// TwinCAT 3 PLC project lamp_lv17_motion
// ProgramVersion: 3.1.4022.7
// libraries:
//   Tc2_MC2, * (Beckhoff Automation GmbH)
//   Tc2_Standard, * (Beckhoff Automation GmbH)
//   Tc2_System, * (Beckhoff Automation GmbH)
//   Tc2_Utilities, * (Beckhoff Automation GmbH)
//   Tc3_Module, * (Beckhoff Automation GmbH)
//   lcls-twincat-motion,newest,SLAC
// project tree:
//   / PlcTask.TcTTO (not stored)
//   POUs/ Main.TcPOU
// real-time tasks:
//   TASK PlcTask: cycle T#10ms, priority 20, ADS port 350
// motion (NC):
//   TASK NC-Task 1 SAF: cycle T#2ms, priority 4, ADS port 501
//   TASK NC-Task 1 SVB: cycle T#10ms, priority 8, ADS port 511
//   AXIS GasJetX (id 1)
//   AXIS GasJetY (id 2)
//   AXIS GasJetZ (id 3)
//   AXIS SamplePaddleX (id 4)
//     Dynamic: Acceleration=2, Deceleration=2, DelayTime=0.008
//     Velo: Maximum=1
//     TargetPosControl: Range=0.001, Time=0.1
//     OtherSettings: AllowMotionCmdToSlave=true
//     encoder EncType=4
//       EncPara: ScaleFactorNumerator=1e-05, Inverse=true, MaxCount=#xffffffff
//         SoftEndMinControl: Range=-39
//         Inc: RefSoftSyncMask=#x0000ffff
//     drive DrvType=24
//       DrvPara: Inverse=true
//         Analog: VeloReferenz=10, ScaleFactorActTorque=0.1
//         TimeComp: TaskDelayCycles=1
//     controller CtrType=2
//       CtrPara: PriorControlFactor=1
//         PosDiffControl: Range=1
//         PID: PosKp=20, PosExtKp=50, DeadBandPosition=0.0005
//         Observer: BandWidth=20
//   AXIS SamplePaddleY (id 5)
//     Dynamic: Acceleration=2, Deceleration=2, DelayTime=0.008
//     Velo: Maximum=1
//     TargetPosControl: Range=0.01, Time=0.1
//     OtherSettings: AllowMotionCmdToSlave=true
//     encoder EncType=4
//       EncPara: ScaleFactorNumerator=2e-05, Inverse=true, MaxCount=#xffffffff
//         SoftEndMinControl: Range=-10
//         SoftEndMaxControl: Range=10
//         Inc: RefSoftSyncMask=#x0000ffff
//     drive DrvType=24
//       DrvPara: Inverse=true
//         Analog: VeloReferenz=5, ScaleFactorActTorque=0.1
//         TimeComp: TaskDelayCycles=1
//     controller CtrType=2
//       CtrPara: PriorControlFactor=1
//         PosDiffControl: Range=0.5
//         PID: PosKp=40, PosExtKp=75, DeadBandPosition=0.0005
//         Observer: BandWidth=20
//   AXIS SamplePaddleZ (id 6)
//     Dynamic: Acceleration=2, Deceleration=2, DelayTime=0.008
//     Velo: Maximum=1
//     TargetPosControl: Range=0.001, Time=0.1
//     OtherSettings: AllowMotionCmdToSlave=true
//     encoder EncType=4
//       EncPara: ScaleFactorNumerator=1e-05, Inverse=true, MaxCount=#xffffffff
//         Inc: RefSoftSyncMask=#x0000ffff
//     drive DrvType=24
//       DrvPara: Inverse=true
//         Analog: VeloReferenz=10, ScaleFactorActTorque=0.1
//         TimeComp: TaskDelayCycles=1
//     controller CtrType=2
//       CtrPara: PriorControlFactor=1
//         PosDiffControl: Range=1
//         PID: PosKp=20, PosExtKp=50, DeadBandPosition=0.0005
//         Observer: BandWidth=20
//   AXIS DetectorX (id 7)
//     Dynamic: Acceleration=2, Deceleration=2
//     Velo: Maximum=1
//     TargetPosControl: Range=0.001
//     OtherSettings: AllowMotionCmdToSlave=true
//     encoder EncType=4
//       EncPara: ScaleFactorNumerator=7.8125e-05, Inverse=true, MaxCount=#x0000ffff
//         Inc: RefSoftSyncMask=#x0000ffff
//     drive DrvType=24
//       DrvPara: Inverse=true
//         Analog: VeloReferenz=10, ScaleFactorActTorque=0.1
//         TimeComp: TaskDelayCycles=1
//     controller CtrType=2
//       CtrPara: PriorControlFactor=1
//         PosDiffControl: Range=1
//         PID: PosKp=20, PosExtKp=50, DeadBandPosition=0.0005
//         Observer: BandWidth=20
//   AXIS DetectorY (id 8)
//     Dynamic: Acceleration=2, Deceleration=2
//     Velo: Maximum=1
//     TargetPosControl: Range=0.001
//     OtherSettings: AllowMotionCmdToSlave=true
//     encoder EncType=4
//       EncPara: ScaleFactorNumerator=7.8125e-05, MaxCount=#x0000ffff
//         Inc: RefSoftSyncMask=#x0000ffff
//     drive DrvType=24
//       Analog: VeloReferenz=10, ScaleFactorActTorque=0.1
//       TimeComp: TaskDelayCycles=1
//     controller CtrType=2
//       CtrPara: PriorControlFactor=1
//         PosDiffControl: Range=1
//         PID: PosKp=20, PosExtKp=50, DeadBandPosition=0.0005
//         Observer: BandWidth=20
// I/O:
//   DEVICE PLC Rail (EtherCAT)
// variable links:
//   (this object) <-> PLC Rail (EtherCAT)/Power (EK1200)/PLC Junction 1 (EK1122)/X1 VacuumMotion (EK1100)/SamplePaddleX-Enc-EL5021
//     Enc/Inputs/In/nDataIn1 <-> ENC Status/Counter value
//     Enc/Inputs/In/nDataIn2 <-> ENC Status/Latch value
//     Enc/Inputs/In/nState1 <-> ENC Status/Status/Latch C valid
//     Enc/Inputs/In/nState1 @bit 2 <-> ENC Status/Status/Set counter done
//     Enc/Inputs/In/nState2 @bit 2 <-> ENC Status/Status/Status of input C
//     Enc/Inputs/In/nState2 @bit 5 <-> ENC Status/Status/Sync error
//     Enc/Inputs/In/nState2 @bit 6 <-> ENC Status/Status/TxPDO State
//     Enc/Inputs/In/nState2 @bit 7 <-> ENC Status/Status/TxPDO Toggle
//     Enc/Inputs/In/nState3 @bit 4 <-> ENC Status/Status/Amplitude error
//     Enc/Inputs/In/nState3 @bit 3 <-> ENC Status/Status/Frequency error
//     Enc/Inputs/In/nState4 @bit 1 <-> WcState/InputToggle
//     Enc/Inputs/In/nState4 <-> WcState/WcState
//     Enc/Outputs/Out/nCtrl1 <-> ENC Control/Control/Enable latch C
//     Enc/Outputs/Out/nCtrl1 @bit 2 <-> ENC Control/Control/Set counter
//     Enc/Outputs/Out/nDataOut1 <-> ENC Control/Set counter value
//   (this object) <-> PLC Rail (EtherCAT)/Power (EK1200)/PLC Junction 1 (EK1122)/X1 VacuumMotion (EK1100)/SamplePaddleX-Mot-EL7041
//     Drive/Inputs/In/nState1 @bit 3 <-> STM Status/Status/Error
//     Drive/Inputs/In/nState1 @bit 5 <-> STM Status/Status/Moving negative
//     Drive/Inputs/In/nState1 @bit 4 <-> STM Status/Status/Moving positive
//     Drive/Inputs/In/nState1 @bit 1 <-> STM Status/Status/Ready
//     Drive/Inputs/In/nState1 <-> STM Status/Status/Ready to enable
//     Drive/Inputs/In/nState1 @bit 6 <-> STM Status/Status/Torque reduced
//     Drive/Inputs/In/nState1 @bit 2 <-> STM Status/Status/Warning
//     Drive/Inputs/In/nState2 @bit 3 <-> STM Status/Status/Digital input 1
//     Drive/Inputs/In/nState2 @bit 4 <-> STM Status/Status/Digital input 2
//     Drive/Inputs/In/nState2 @bit 5 <-> STM Status/Status/Sync error
//     Drive/Inputs/In/nState2 @bit 7 <-> STM Status/Status/TxPDO Toggle
//     Drive/Inputs/In/nState4 @bit 1 <-> WcState/InputToggle
//     Drive/Inputs/In/nState4 <-> WcState/WcState
//     Drive/Outputs/Out/nCtrl1 <-> STM Control/Control/Enable
//     Drive/Outputs/Out/nCtrl1 @bit 2 <-> STM Control/Control/Reduce torque
//     Drive/Outputs/Out/nCtrl1 @bit 1 <-> STM Control/Control/Reset
//     Drive/Outputs/Out/nDataOut2[0] <-> STM Velocity/Velocity
//   (this object) <-> PLC Rail (EtherCAT)/Power (EK1200)/PLC Junction 1 (EK1122)/X1 VacuumMotion (EK1100)/SamplePaddleY-Enc-EL5021
//     Enc/Inputs/In/nDataIn1 <-> ENC Status/Counter value
//     Enc/Inputs/In/nDataIn2 <-> ENC Status/Latch value
//     Enc/Inputs/In/nState1 <-> ENC Status/Status/Latch C valid
//     Enc/Inputs/In/nState1 @bit 2 <-> ENC Status/Status/Set counter done
//     Enc/Inputs/In/nState2 @bit 2 <-> ENC Status/Status/Status of input C
//     Enc/Inputs/In/nState2 @bit 5 <-> ENC Status/Status/Sync error
//     Enc/Inputs/In/nState2 @bit 6 <-> ENC Status/Status/TxPDO State
//     Enc/Inputs/In/nState2 @bit 7 <-> ENC Status/Status/TxPDO Toggle
//     Enc/Inputs/In/nState3 @bit 4 <-> ENC Status/Status/Amplitude error
//     Enc/Inputs/In/nState3 @bit 3 <-> ENC Status/Status/Frequency error
//     Enc/Inputs/In/nState4 @bit 1 <-> WcState/InputToggle
//     Enc/Inputs/In/nState4 <-> WcState/WcState
//     Enc/Outputs/Out/nCtrl1 <-> ENC Control/Control/Enable latch C
//     Enc/Outputs/Out/nCtrl1 @bit 2 <-> ENC Control/Control/Set counter
//     Enc/Outputs/Out/nDataOut1 <-> ENC Control/Set counter value
//   (this object) <-> PLC Rail (EtherCAT)/Power (EK1200)/PLC Junction 1 (EK1122)/X1 VacuumMotion (EK1100)/SamplePaddleY-Mot-EL7041
//     Drive/Inputs/In/nState1 @bit 3 <-> STM Status/Status/Error
//     Drive/Inputs/In/nState1 @bit 5 <-> STM Status/Status/Moving negative
//     Drive/Inputs/In/nState1 @bit 4 <-> STM Status/Status/Moving positive
//     Drive/Inputs/In/nState1 @bit 1 <-> STM Status/Status/Ready
//     Drive/Inputs/In/nState1 <-> STM Status/Status/Ready to enable
//     Drive/Inputs/In/nState1 @bit 6 <-> STM Status/Status/Torque reduced
//     Drive/Inputs/In/nState1 @bit 2 <-> STM Status/Status/Warning
//     Drive/Inputs/In/nState2 @bit 3 <-> STM Status/Status/Digital input 1
//     Drive/Inputs/In/nState2 @bit 4 <-> STM Status/Status/Digital input 2
//     Drive/Inputs/In/nState2 @bit 5 <-> STM Status/Status/Sync error
//     Drive/Inputs/In/nState2 @bit 7 <-> STM Status/Status/TxPDO Toggle
//     Drive/Inputs/In/nState4 @bit 1 <-> WcState/InputToggle
//     Drive/Inputs/In/nState4 <-> WcState/WcState
//     Drive/Outputs/Out/nCtrl1 <-> STM Control/Control/Enable
//     Drive/Outputs/Out/nCtrl1 @bit 2 <-> STM Control/Control/Reduce torque
//     Drive/Outputs/Out/nCtrl1 @bit 1 <-> STM Control/Control/Reset
//     Drive/Outputs/Out/nDataOut2[0] <-> STM Velocity/Velocity
//   (this object) <-> PLC Rail (EtherCAT)/Power (EK1200)/PLC Junction 1 (EK1122)/X1 VacuumMotion (EK1100)/SamplePaddleZ-Enc-EL5021
//     Enc/Inputs/In/nDataIn1 <-> ENC Status/Counter value
//     Enc/Inputs/In/nDataIn2 <-> ENC Status/Latch value
//     Enc/Inputs/In/nState1 <-> ENC Status/Status/Latch C valid
//     Enc/Inputs/In/nState1 @bit 2 <-> ENC Status/Status/Set counter done
//     Enc/Inputs/In/nState2 @bit 2 <-> ENC Status/Status/Status of input C
//     Enc/Inputs/In/nState2 @bit 5 <-> ENC Status/Status/Sync error
//     Enc/Inputs/In/nState2 @bit 6 <-> ENC Status/Status/TxPDO State
//     Enc/Inputs/In/nState2 @bit 7 <-> ENC Status/Status/TxPDO Toggle
//     Enc/Inputs/In/nState3 @bit 4 <-> ENC Status/Status/Amplitude error
//     Enc/Inputs/In/nState3 @bit 3 <-> ENC Status/Status/Frequency error
//     Enc/Inputs/In/nState4 @bit 1 <-> WcState/InputToggle
//     Enc/Inputs/In/nState4 <-> WcState/WcState
//     Enc/Outputs/Out/nCtrl1 <-> ENC Control/Control/Enable latch C
//     Enc/Outputs/Out/nCtrl1 @bit 2 <-> ENC Control/Control/Set counter
//     Enc/Outputs/Out/nDataOut1 <-> ENC Control/Set counter value
//   (this object) <-> PLC Rail (EtherCAT)/Power (EK1200)/PLC Junction 1 (EK1122)/X1 VacuumMotion (EK1100)/SamplePaddleZ-Mot-EL7041
//     Drive/Inputs/In/nState1 @bit 3 <-> STM Status/Status/Error
//     Drive/Inputs/In/nState1 @bit 5 <-> STM Status/Status/Moving negative
//     Drive/Inputs/In/nState1 @bit 4 <-> STM Status/Status/Moving positive
//     Drive/Inputs/In/nState1 @bit 1 <-> STM Status/Status/Ready
//     Drive/Inputs/In/nState1 <-> STM Status/Status/Ready to enable
//     Drive/Inputs/In/nState1 @bit 6 <-> STM Status/Status/Torque reduced
//     Drive/Inputs/In/nState1 @bit 2 <-> STM Status/Status/Warning
//     Drive/Inputs/In/nState2 @bit 3 <-> STM Status/Status/Digital input 1
//     Drive/Inputs/In/nState2 @bit 4 <-> STM Status/Status/Digital input 2
//     Drive/Inputs/In/nState2 @bit 5 <-> STM Status/Status/Sync error
//     Drive/Inputs/In/nState2 @bit 7 <-> STM Status/Status/TxPDO Toggle
//     Drive/Inputs/In/nState4 @bit 1 <-> WcState/InputToggle
//     Drive/Inputs/In/nState4 <-> WcState/WcState
//     Drive/Outputs/Out/nCtrl1 <-> STM Control/Control/Enable
//     Drive/Outputs/Out/nCtrl1 @bit 2 <-> STM Control/Control/Reduce torque
//     Drive/Outputs/Out/nCtrl1 @bit 1 <-> STM Control/Control/Reset
//     Drive/Outputs/Out/nDataOut2[0] <-> STM Velocity/Velocity
//   (this object) <-> PLC Rail (EtherCAT)/Power (EK1200)/PLC Junction 1 (EK1122)/X1 VacuumMotion (EK1100)/DetectorX-Mot-EL7041
//     Drive/Inputs/In/nState1 @bit 3 <-> STM Status/Status/Error
//     Drive/Inputs/In/nState1 @bit 5 <-> STM Status/Status/Moving negative
//     Drive/Inputs/In/nState1 @bit 4 <-> STM Status/Status/Moving positive
//     Drive/Inputs/In/nState1 @bit 1 <-> STM Status/Status/Ready
//     Drive/Inputs/In/nState1 <-> STM Status/Status/Ready to enable
//     Drive/Inputs/In/nState1 @bit 6 <-> STM Status/Status/Torque reduced
//     Drive/Inputs/In/nState1 @bit 2 <-> STM Status/Status/Warning
//     Drive/Inputs/In/nState2 @bit 3 <-> STM Status/Status/Digital input 1
//     Drive/Inputs/In/nState2 @bit 4 <-> STM Status/Status/Digital input 2
//     Drive/Inputs/In/nState2 @bit 5 <-> STM Status/Status/Sync error
//     Drive/Inputs/In/nState2 @bit 7 <-> STM Status/Status/TxPDO Toggle
//     Drive/Inputs/In/nState4 @bit 1 <-> WcState/InputToggle
//     Drive/Inputs/In/nState4 <-> WcState/WcState
//     Drive/Outputs/Out/nCtrl1 <-> STM Control/Control/Enable
//     Drive/Outputs/Out/nCtrl1 @bit 2 <-> STM Control/Control/Reduce torque
//     Drive/Outputs/Out/nCtrl1 @bit 1 <-> STM Control/Control/Reset
//     Drive/Outputs/Out/nDataOut2[0] <-> STM Velocity/Velocity
//     Enc/Inputs/In/nDataIn1[0] <-> ENC Status compact/Counter value
//     Enc/Inputs/In/nDataIn2[0] <-> ENC Status compact/Latch value
//     Enc/Inputs/In/nState1 @bit 4 <-> ENC Status compact/Status/Counter overflow
//     Enc/Inputs/In/nState1 @bit 3 <-> ENC Status compact/Status/Counter underflow
//     Enc/Inputs/In/nState1 @bit 7 <-> ENC Status compact/Status/Extrapolation stall
//     Enc/Inputs/In/nState1 <-> ENC Status compact/Status/Latch C valid
//     Enc/Inputs/In/nState1 @bit 1 <-> ENC Status compact/Status/Latch extern valid
//     Enc/Inputs/In/nState1 @bit 2 <-> ENC Status compact/Status/Set counter done
//     Enc/Inputs/In/nState2 @bit 4 <-> ENC Status compact/Status/Status of extern latch
//     Enc/Inputs/In/nState2 <-> ENC Status compact/Status/Status of input A
//     Enc/Inputs/In/nState2 @bit 1 <-> ENC Status compact/Status/Status of input B
//     Enc/Inputs/In/nState2 @bit 2 <-> ENC Status compact/Status/Status of input C
//     Enc/Inputs/In/nState2 @bit 5 <-> ENC Status compact/Status/Sync error
//     Enc/Inputs/In/nState2 @bit 7 <-> ENC Status compact/Status/TxPDO Toggle
//     Enc/Inputs/In/nState4 @bit 1 <-> WcState/InputToggle
//     Enc/Inputs/In/nState4 <-> WcState/WcState
//     Enc/Outputs/Out/nCtrl1 <-> ENC Control compact/Control/Enable latch C
//     Enc/Outputs/Out/nCtrl1 @bit 3 <-> ENC Control compact/Control/Enable latch extern on negative edge
//     Enc/Outputs/Out/nCtrl1 @bit 1 <-> ENC Control compact/Control/Enable latch extern on positive edge
//     Enc/Outputs/Out/nCtrl1 @bit 2 <-> ENC Control compact/Control/Set counter
//     Enc/Outputs/Out/nDataOut1[0] <-> ENC Control compact/Set counter value
//   (this object) <-> PLC Rail (EtherCAT)/Power (EK1200)/PLC Junction 1 (EK1122)/X1 VacuumMotion (EK1100)/DetectorY-Mot-EL7041
//     Drive/Inputs/In/nState1 @bit 3 <-> STM Status/Status/Error
//     Drive/Inputs/In/nState1 @bit 5 <-> STM Status/Status/Moving negative
//     Drive/Inputs/In/nState1 @bit 4 <-> STM Status/Status/Moving positive
//     Drive/Inputs/In/nState1 @bit 1 <-> STM Status/Status/Ready
//     Drive/Inputs/In/nState1 <-> STM Status/Status/Ready to enable
//     Drive/Inputs/In/nState1 @bit 6 <-> STM Status/Status/Torque reduced
//     Drive/Inputs/In/nState1 @bit 2 <-> STM Status/Status/Warning
//     Drive/Inputs/In/nState2 @bit 3 <-> STM Status/Status/Digital input 1
//     Drive/Inputs/In/nState2 @bit 4 <-> STM Status/Status/Digital input 2
//     Drive/Inputs/In/nState2 @bit 5 <-> STM Status/Status/Sync error
//     Drive/Inputs/In/nState2 @bit 7 <-> STM Status/Status/TxPDO Toggle
//     Drive/Inputs/In/nState4 @bit 1 <-> WcState/InputToggle
//     Drive/Inputs/In/nState4 <-> WcState/WcState
//     Drive/Outputs/Out/nCtrl1 <-> STM Control/Control/Enable
//     Drive/Outputs/Out/nCtrl1 @bit 2 <-> STM Control/Control/Reduce torque
//     Drive/Outputs/Out/nCtrl1 @bit 1 <-> STM Control/Control/Reset
//     Drive/Outputs/Out/nDataOut2[0] <-> STM Velocity/Velocity
//     Enc/Inputs/In/nDataIn1[0] <-> ENC Status compact/Counter value
//     Enc/Inputs/In/nDataIn2[0] <-> ENC Status compact/Latch value
//     Enc/Inputs/In/nState1 @bit 4 <-> ENC Status compact/Status/Counter overflow
//     Enc/Inputs/In/nState1 @bit 3 <-> ENC Status compact/Status/Counter underflow
//     Enc/Inputs/In/nState1 @bit 7 <-> ENC Status compact/Status/Extrapolation stall
//     Enc/Inputs/In/nState1 <-> ENC Status compact/Status/Latch C valid
//     Enc/Inputs/In/nState1 @bit 1 <-> ENC Status compact/Status/Latch extern valid
//     Enc/Inputs/In/nState1 @bit 2 <-> ENC Status compact/Status/Set counter done
//     Enc/Inputs/In/nState2 @bit 4 <-> ENC Status compact/Status/Status of extern latch
//     Enc/Inputs/In/nState2 <-> ENC Status compact/Status/Status of input A
//     Enc/Inputs/In/nState2 @bit 1 <-> ENC Status compact/Status/Status of input B
//     Enc/Inputs/In/nState2 @bit 2 <-> ENC Status compact/Status/Status of input C
//     Enc/Inputs/In/nState2 @bit 5 <-> ENC Status compact/Status/Sync error
//     Enc/Inputs/In/nState2 @bit 7 <-> ENC Status compact/Status/TxPDO Toggle
//     Enc/Inputs/In/nState4 @bit 1 <-> WcState/InputToggle
//     Enc/Inputs/In/nState4 <-> WcState/WcState
//     Enc/Outputs/Out/nCtrl1 <-> ENC Control compact/Control/Enable latch C
//     Enc/Outputs/Out/nCtrl1 @bit 3 <-> ENC Control compact/Control/Enable latch extern on negative edge
//     Enc/Outputs/Out/nCtrl1 @bit 1 <-> ENC Control compact/Control/Enable latch extern on positive edge
//     Enc/Outputs/Out/nCtrl1 @bit 2 <-> ENC Control compact/Control/Set counter
//     Enc/Outputs/Out/nDataOut1[0] <-> ENC Control compact/Set counter value
//   lamp_lv17_motion Instance <-> PLC Rail (EtherCAT)/Power (EK1200)/PLC Junction 1 (EK1122)/X1 AtmosphereMotion (EK1100)/GasJetX-EL7041
//     PlcTask Inputs/Main.M1.bLimitBackwardEnable <-> STM Status/Status/Digital input 2
//     PlcTask Inputs/Main.M1.bLimitForwardEnable <-> STM Status/Status/Digital input 1
//   lamp_lv17_motion Instance <-> PLC Rail (EtherCAT)/Power (EK1200)/PLC Junction 1 (EK1122)/X1 AtmosphereMotion (EK1100)/GasJetY-EL7041
//     PlcTask Inputs/Main.M2.bLimitBackwardEnable <-> STM Status/Status/Digital input 2
//     PlcTask Inputs/Main.M2.bLimitForwardEnable <-> STM Status/Status/Digital input 1
//   lamp_lv17_motion Instance <-> PLC Rail (EtherCAT)/Power (EK1200)/PLC Junction 1 (EK1122)/X1 AtmosphereMotion (EK1100)/GasJetZ-EL7041
//     PlcTask Inputs/Main.M3.bLimitBackwardEnable <-> STM Status/Status/Digital input 2
//     PlcTask Inputs/Main.M3.bLimitForwardEnable <-> STM Status/Status/Digital input 1
//   lamp_lv17_motion Instance <-> PLC Rail (EtherCAT)/Power (EK1200)/PLC Junction 1 (EK1122)/X1 VacuumMotion (EK1100)/DetectorXY-Limits-EL1084
//     PlcTask Inputs/Main.M7.bLimitBackwardEnable <-> Channel 2/Input
//     PlcTask Inputs/Main.M8.bLimitBackwardEnable <-> Channel 4/Input
//     PlcTask Inputs/Main.M7.bLimitForwardEnable <-> Channel 1/Input
//   lamp_lv17_motion Instance <-> PLC Rail (EtherCAT)/Power (EK1200)/PLC Junction 1 (EK1122)/X1 VacuumMotion (EK1100)/SamplePaddleXY-Limits-EL1084
//     PlcTask Inputs/Main.M4.bLimitBackwardEnable <-> Channel 2/Input
//     PlcTask Inputs/Main.M5.bLimitBackwardEnable <-> Channel 3/Input
//     PlcTask Inputs/Main.M4.bLimitForwardEnable <-> Channel 1/Input
//     PlcTask Inputs/Main.M5.bLimitForwardEnable <-> Channel 4/Input
//   lamp_lv17_motion Instance <-> PLC Rail (EtherCAT)/Power (EK1200)/PLC Junction 1 (EK1122)/X1 VacuumMotion (EK1100)/SamplePaddleZ-Limits-EL1084
//     PlcTask Inputs/Main.M6.bLimitBackwardEnable <-> Channel 2/Input
//     PlcTask Inputs/Main.M6.bLimitForwardEnable <-> Channel 1/Input
//   lamp_lv17_motion Instance <-> NC-Task 1 SAF/Axes/DetectorX
//     PlcTask Inputs/Main.M7.Axis.NcToPlc <-> Outputs/ToPlc
//     PlcTask Outputs/Main.M7.Axis.PlcToNc <-> Inputs/FromPlc
//   lamp_lv17_motion Instance <-> NC-Task 1 SAF/Axes/DetectorY
//     PlcTask Inputs/Main.M8.Axis.NcToPlc <-> Outputs/ToPlc
//     PlcTask Outputs/Main.M8.Axis.PlcToNc <-> Inputs/FromPlc
//   lamp_lv17_motion Instance <-> NC-Task 1 SAF/Axes/GasJetX
//     PlcTask Inputs/Main.M1.Axis.NcToPlc <-> Outputs/ToPlc
//     PlcTask Outputs/Main.M1.Axis.PlcToNc <-> Inputs/FromPlc
//   lamp_lv17_motion Instance <-> NC-Task 1 SAF/Axes/GasJetY
//     PlcTask Inputs/Main.M2.Axis.NcToPlc <-> Outputs/ToPlc
//     PlcTask Outputs/Main.M2.Axis.PlcToNc <-> Inputs/FromPlc
//   lamp_lv17_motion Instance <-> NC-Task 1 SAF/Axes/GasJetZ
//     PlcTask Inputs/Main.M3.Axis.NcToPlc <-> Outputs/ToPlc
//     PlcTask Outputs/Main.M3.Axis.PlcToNc <-> Inputs/FromPlc
//   lamp_lv17_motion Instance <-> NC-Task 1 SAF/Axes/SamplePaddleX
//     PlcTask Inputs/Main.M4.Axis.NcToPlc <-> Outputs/ToPlc
//     PlcTask Outputs/Main.M4.Axis.PlcToNc <-> Inputs/FromPlc
//   lamp_lv17_motion Instance <-> NC-Task 1 SAF/Axes/SamplePaddleY
//     PlcTask Inputs/Main.M5.Axis.NcToPlc <-> Outputs/ToPlc
//     PlcTask Outputs/Main.M5.Axis.PlcToNc <-> Inputs/FromPlc
//   lamp_lv17_motion Instance <-> NC-Task 1 SAF/Axes/SamplePaddleZ
//     PlcTask Inputs/Main.M6.Axis.NcToPlc <-> Outputs/ToPlc
//     PlcTask Outputs/Main.M6.Axis.PlcToNc <-> Inputs/FromPlc

// ---- POUs/Main.TcPOU
PROGRAM Main
VAR
	// Motors
	{attribute 'TcLinkTo' := '.bLimitForwardEnable:=TIIB[GasJetX-EL7041]^STM Status^Status^Digital input 1;
                              .bLimitBackwardEnable:=TIIB[GasJetX-EL7041]^STM Status^Status^Digital input 2'}
	{attribute 'pytmc' := '
		pv: TMO:LAMP:MMS:01
	'}
	M1 		: DUT_MotionStage := (bPowerSelf:=TRUE, 
    nEnableMode:=ENUM_StageEnableMode.DURING_MOTION,
//    nEnableMode:=ENUM_StageEnableMode.ALWAYS,
    nHomingMode := ENUM_EpicsHomeCmd.ABSOLUTE_SET ); // Gas Jet X

	{attribute 'TcLinkTo' := '.bLimitForwardEnable:=TIIB[GasJetY-EL7041]^STM Status^Status^Digital input 1;
                              .bLimitBackwardEnable:=TIIB[GasJetY-EL7041]^STM Status^Status^Digital input 2'}
	{attribute 'pytmc' := '
		pv: TMO:LAMP:MMS:02
	'}
	M2		: DUT_MotionStage := (bPowerSelf:=TRUE, 
    nEnableMode:=ENUM_StageEnableMode.DURING_MOTION,
//    nEnableMode:=ENUM_StageEnableMode.ALWAYS,
    nHomingMode := ENUM_EpicsHomeCmd.ABSOLUTE_SET); // Gas Jet Y

	{attribute 'TcLinkTo' := '.bLimitForwardEnable:=TIIB[GasJetZ-EL7041]^STM Status^Status^Digital input 1;
                              .bLimitBackwardEnable:=TIIB[GasJetZ-EL7041]^STM Status^Status^Digital input 2'}
	{attribute 'pytmc' := '
		pv: TMO:LAMP:MMS:03
	'}
	M3		: DUT_MotionStage := (bPowerSelf:=TRUE, 
    nEnableMode:=ENUM_StageEnableMode.DURING_MOTION,
//    nEnableMode:=ENUM_StageEnableMode.ALWAYS,
    nHomingMode := ENUM_EpicsHomeCmd.ABSOLUTE_SET); // Gas Jet Z

	{attribute 'TcLinkTo' := '.bLimitForwardEnable:=TIIB[SamplePaddleXY-Limits-EL1084]^Channel 1^Input;
                              .bLimitBackwardEnable:=TIIB[SamplePaddleXY-Limits-EL1084]^Channel 2^Input'}
	{attribute 'pytmc' := '
		pv: TMO:LAMP:MMS:04
	'}
	M4  	: DUT_MotionStage := (bPowerSelf:=TRUE, 
    nEnableMode:=ENUM_StageEnableMode.DURING_MOTION,
//    nEnableMode:=ENUM_StageEnableMode.ALWAYS,
    nHomingMode := ENUM_EpicsHomeCmd.ABSOLUTE_SET); // Sample Paddle X

	{attribute 'TcLinkTo' := '.bLimitForwardEnable:=TIIB[SamplePaddleXY-Limits-EL1084]^Channel 4^Input;
                              .bLimitBackwardEnable:=TIIB[SamplePaddleXY-Limits-EL1084]^Channel 3^Input'}
	{attribute 'pytmc' := '
		pv: TMO:LAMP:MMS:05
	'}
	M5  	: DUT_MotionStage := (bPowerSelf:=TRUE, 
    nEnableMode:=ENUM_StageEnableMode.DURING_MOTION,
//    nEnableMode:=ENUM_StageEnableMode.ALWAYS,
    nHomingMode := ENUM_EpicsHomeCmd.ABSOLUTE_SET); // Sample Paddle Y

	{attribute 'TcLinkTo' := '.bLimitForwardEnable:=TIIB[SamplePaddleZ-Limits-EL1084]^Channel 1^Input;
                              .bLimitBackwardEnable:=TIIB[SamplePaddleZ-Limits-EL1084]^Channel 2^Input'}
	{attribute 'pytmc' := '
		pv: TMO:LAMP:MMS:06
    '}
	M6  	: DUT_MotionStage := (bPowerSelf:=TRUE, 
    nEnableMode:=ENUM_StageEnableMode.DURING_MOTION,
//    nEnableMode:=ENUM_StageEnableMode.ALWAYS,
    nHomingMode := ENUM_EpicsHomeCmd.ABSOLUTE_SET); // Sample Paddle Z
	
	{attribute 'TcLinkTo' := '.bLimitForwardEnable:=TIIB[DetectorXY-Limits-EL1084]^Channel 1^Input;
                              .bLimitBackwardEnable:=TIIB[DetectorXY-Limits-EL1084]^Channel 2^Input'}
	{attribute 'pytmc' := '
		pv: TMO:LAMP:MMS:07
    '}
	M7  	: DUT_MotionStage := (bPowerSelf:=TRUE, 
    nEnableMode:=ENUM_StageEnableMode.DURING_MOTION,
//    nEnableMode:=ENUM_StageEnableMode.ALWAYS,
    nHomingMode := ENUM_EpicsHomeCmd.ABSOLUTE_SET); // Detector X
	
	{attribute 'TcLinkTo' := '.bLimitBackwardEnable:=TIIB[DetectorXY-Limits-EL1084]^Channel 4^Input'}
	// .bLimitForwardEnable:=TIIB[DetectorXY-Limits-EL1084]^Channel 3^Input;
	
	//             Lim+ wire is not terminated correctly on vacuum side,
    //             scientists will use software limits and camera-guided motion)
	
	{attribute 'pytmc' := '
		pv: TMO:LAMP:MMS:08
    '}
	M8  	: DUT_MotionStage := (bPowerSelf:=TRUE, 
    nEnableMode:=ENUM_StageEnableMode.DURING_MOTION,
//    nEnableMode:=ENUM_StageEnableMode.ALWAYS,
    nHomingMode := ENUM_EpicsHomeCmd.ABSOLUTE_SET); // Detector Y
	
	
	fbMotionStageM1	: FB_MotionStage;
	fbMotionStageM2	: FB_MotionStage;
	fbMotionStageM3	: FB_MotionStage;
	fbMotionStageM4	: FB_MotionStage;
	fbMotionStageM5	: FB_MotionStage;
	fbMotionStageM6	: FB_MotionStage;
	fbMotionStageM7	: FB_MotionStage;
	fbMotionStageM8	: FB_MotionStage;
END_VAR

	// Hardware Enable
	// Gas Jet
	M1.bHardwareEnable	:= TRUE;
	M2.bHardwareEnable	:= TRUE;
	M3.bHardwareEnable	:= TRUE;
	// Sample Paddle
	M4.bHardwareEnable	:= TRUE;
	M5.bHardwareEnable	:= TRUE;
	M6.bHardwareEnable	:= TRUE;
	// Detector (Epix-100)
	M7.bHardwareEnable	:= TRUE;
	M8.bHardwareEnable	:= TRUE;
	
	// Detector X (Lim+ wire is not terminated correctly on vacuum side,
    //             scientists will use software limits and camera-guided motion)
	M7.bLimitForwardEnable := True;
	M7.bLimitBackwardEnable := True;
	// fbMotionStage
	// Gas Jet
	fbMotionStageM1(stMotionStage:=M1);
	fbMotionStageM2(stMotionStage:=M2);
	fbMotionStageM3(stMotionStage:=M3);
	// Sample Paddle
	fbMotionStageM4(stMotionStage:=M4);
	fbMotionStageM5(stMotionStage:=M5);
	fbMotionStageM6(stMotionStage:=M6);
	// Detector (Epix-100)
	fbMotionStageM7(stMotionStage:=M7);
	fbMotionStageM8(stMotionStage:=M8);

END_PROGRAM
